VAR_GLOBAL CONSTANT
	cintMaxCharge: INT := 10;
END_VAR

(* stored: Version 1.1.0.1, ProductVersion 3.1.0.19
   GVL Const_HPS: Id {3fee818e-bba7-4c75-be5f-3303d926f516} *)
